PROGRAM ClangsonicUSModbusFeedbackCtrl
VAR
	ARfbUs: ARRAY [1..12] OF fbRawRatioConversionUsPercent;

END_VAR

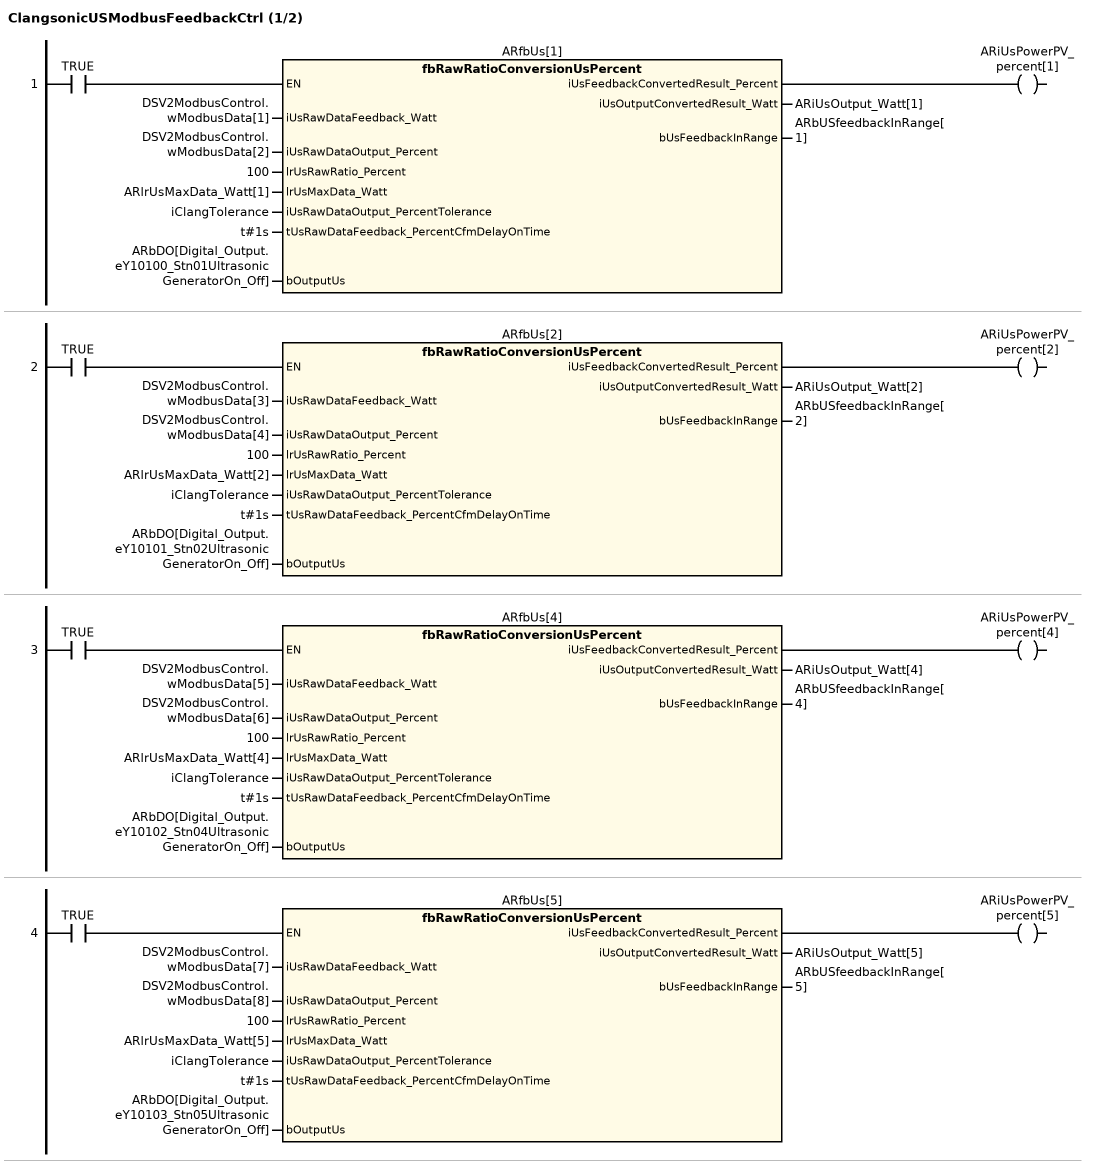
// NETWORK 1
ARfbUs[1](
    iUsRawDataFeedback_Watt := DSV2ModbusControl.wModbusData[1],
    iUsRawDataOutput_Percent := DSV2ModbusControl.wModbusData[2],
    lrUsRawRatio_Percent := 100,
    lrUsMaxData_Watt := ARlrUsMaxData_Watt[1],
    iUsRawDataOutput_PercentTolerance := iClangTolerance,
    tUsRawDataFeedback_PercentCfmDelayOnTime := t#1s,
    bOutputUs := ARbDO[Digital_Output.eY10100_Stn01UltrasonicGeneratorOn_Off],
    iUsOutputConvertedResult_Watt => ARiUsOutput_Watt[1],
    bUsFeedbackInRange => ARbUSfeedbackInRange[1]); // fbRawRatioConversionUsPercent
ARiUsPowerPV_percent[1] := ARfbUs[1].iUsFeedbackConvertedResult_Percent;

// NETWORK 2
ARfbUs[2](
    iUsRawDataFeedback_Watt := DSV2ModbusControl.wModbusData[3],
    iUsRawDataOutput_Percent := DSV2ModbusControl.wModbusData[4],
    lrUsRawRatio_Percent := 100,
    lrUsMaxData_Watt := ARlrUsMaxData_Watt[2],
    iUsRawDataOutput_PercentTolerance := iClangTolerance,
    tUsRawDataFeedback_PercentCfmDelayOnTime := t#1s,
    bOutputUs := ARbDO[Digital_Output.eY10101_Stn02UltrasonicGeneratorOn_Off],
    iUsOutputConvertedResult_Watt => ARiUsOutput_Watt[2],
    bUsFeedbackInRange => ARbUSfeedbackInRange[2]); // fbRawRatioConversionUsPercent
ARiUsPowerPV_percent[2] := ARfbUs[2].iUsFeedbackConvertedResult_Percent;

// NETWORK 3
ARfbUs[4](
    iUsRawDataFeedback_Watt := DSV2ModbusControl.wModbusData[5],
    iUsRawDataOutput_Percent := DSV2ModbusControl.wModbusData[6],
    lrUsRawRatio_Percent := 100,
    lrUsMaxData_Watt := ARlrUsMaxData_Watt[4],
    iUsRawDataOutput_PercentTolerance := iClangTolerance,
    tUsRawDataFeedback_PercentCfmDelayOnTime := t#1s,
    bOutputUs := ARbDO[Digital_Output.eY10102_Stn04UltrasonicGeneratorOn_Off],
    iUsOutputConvertedResult_Watt => ARiUsOutput_Watt[4],
    bUsFeedbackInRange => ARbUSfeedbackInRange[4]); // fbRawRatioConversionUsPercent
ARiUsPowerPV_percent[4] := ARfbUs[4].iUsFeedbackConvertedResult_Percent;

// NETWORK 4
ARfbUs[5](
    iUsRawDataFeedback_Watt := DSV2ModbusControl.wModbusData[7],
    iUsRawDataOutput_Percent := DSV2ModbusControl.wModbusData[8],
    lrUsRawRatio_Percent := 100,
    lrUsMaxData_Watt := ARlrUsMaxData_Watt[5],
    iUsRawDataOutput_PercentTolerance := iClangTolerance,
    tUsRawDataFeedback_PercentCfmDelayOnTime := t#1s,
    bOutputUs := ARbDO[Digital_Output.eY10103_Stn05UltrasonicGeneratorOn_Off],
    iUsOutputConvertedResult_Watt => ARiUsOutput_Watt[5],
    bUsFeedbackInRange => ARbUSfeedbackInRange[5]); // fbRawRatioConversionUsPercent
ARiUsPowerPV_percent[5] := ARfbUs[5].iUsFeedbackConvertedResult_Percent;

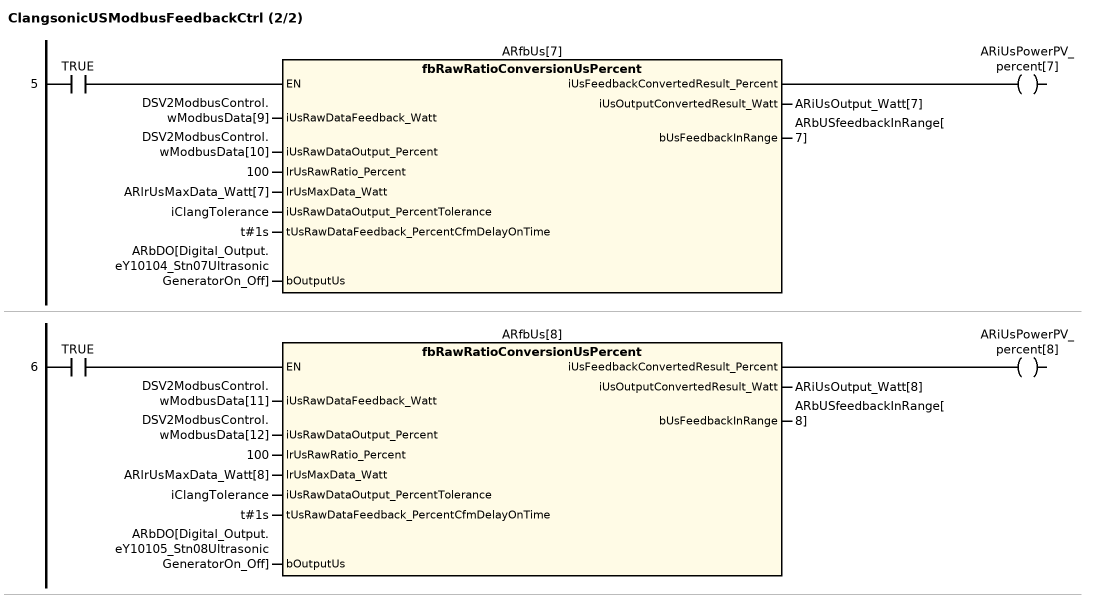
// NETWORK 5
ARfbUs[7](
    iUsRawDataFeedback_Watt := DSV2ModbusControl.wModbusData[9],
    iUsRawDataOutput_Percent := DSV2ModbusControl.wModbusData[10],
    lrUsRawRatio_Percent := 100,
    lrUsMaxData_Watt := ARlrUsMaxData_Watt[7],
    iUsRawDataOutput_PercentTolerance := iClangTolerance,
    tUsRawDataFeedback_PercentCfmDelayOnTime := t#1s,
    bOutputUs := ARbDO[Digital_Output.eY10104_Stn07UltrasonicGeneratorOn_Off],
    iUsOutputConvertedResult_Watt => ARiUsOutput_Watt[7],
    bUsFeedbackInRange => ARbUSfeedbackInRange[7]); // fbRawRatioConversionUsPercent
ARiUsPowerPV_percent[7] := ARfbUs[7].iUsFeedbackConvertedResult_Percent;

// NETWORK 6
ARfbUs[8](
    iUsRawDataFeedback_Watt := DSV2ModbusControl.wModbusData[11],
    iUsRawDataOutput_Percent := DSV2ModbusControl.wModbusData[12],
    lrUsRawRatio_Percent := 100,
    lrUsMaxData_Watt := ARlrUsMaxData_Watt[8],
    iUsRawDataOutput_PercentTolerance := iClangTolerance,
    tUsRawDataFeedback_PercentCfmDelayOnTime := t#1s,
    bOutputUs := ARbDO[Digital_Output.eY10105_Stn08UltrasonicGeneratorOn_Off],
    iUsOutputConvertedResult_Watt => ARiUsOutput_Watt[8],
    bUsFeedbackInRange => ARbUSfeedbackInRange[8]); // fbRawRatioConversionUsPercent
ARiUsPowerPV_percent[8] := ARfbUs[8].iUsFeedbackConvertedResult_Percent;

END_PROGRAM

(* stored: Version 1.1.0.1, ProductVersion 3.1.4024.12
   POU ClangsonicUSModbusFeedbackCtrl: Id {1597cd6f-556c-472d-a4cb-e8fd335e4724}, SpecialFunc None *)
